// Mitsubishi GX Works2 project: EXAM2   PLC: Q03UDV

PROGRAM MAIN
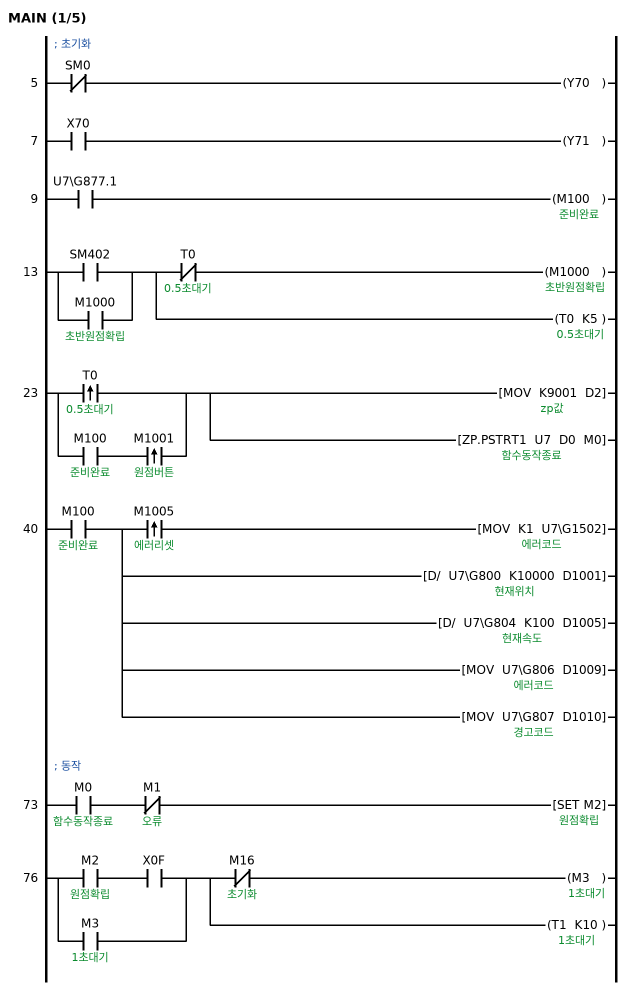
; 초기화
5     LDI     SM0
      OUT     Y70
7     LD      X70
      OUT     Y71
9     LD      U7\G877.1
      OUT     M100  ; 준비완료
13    LD      SM402
      OR      M1000  ; 초반원점확립
      MPS
      ANI     T0  ; 0.5초대기
      OUT     M1000  ; 초반원점확립
      MPP
      OUT     T0 K5  ; 0.5초대기
23    LDP     T0  ; 0.5초대기
      LD      M100  ; 준비완료
      ANDP    M1001  ; 원점버튼
      ORB
      MOV     K9001 D2  ; zp값
      ZP.PSTRT1 U7 D0 M0  ; 함수동작종료
40    LD      M100  ; 준비완료
      MPS
      ANDP    M1005  ; 에러리셋
      MOV     K1 U7\G1502  ; 에러코드
      MPP
      D/      U7\G800 K10000 D1001  ; 현재위치
      D/      U7\G804 K100 D1005  ; 현재속도
      MOV     U7\G806 D1009  ; 에러코드
      MOV     U7\G807 D1010  ; 경고코드
; 동작
73    LD      M0  ; 함수동작종료
      ANI     M1  ; 오류
      SET     M2  ; 원점확립
76    LD      M2  ; 원점확립
      AND     X0F
      OR      M3  ; 1초대기
      MPS
      ANI     M16  ; 초기화
      OUT     M3  ; 1초대기
      MPP
      OUT     T1 K10  ; 1초대기
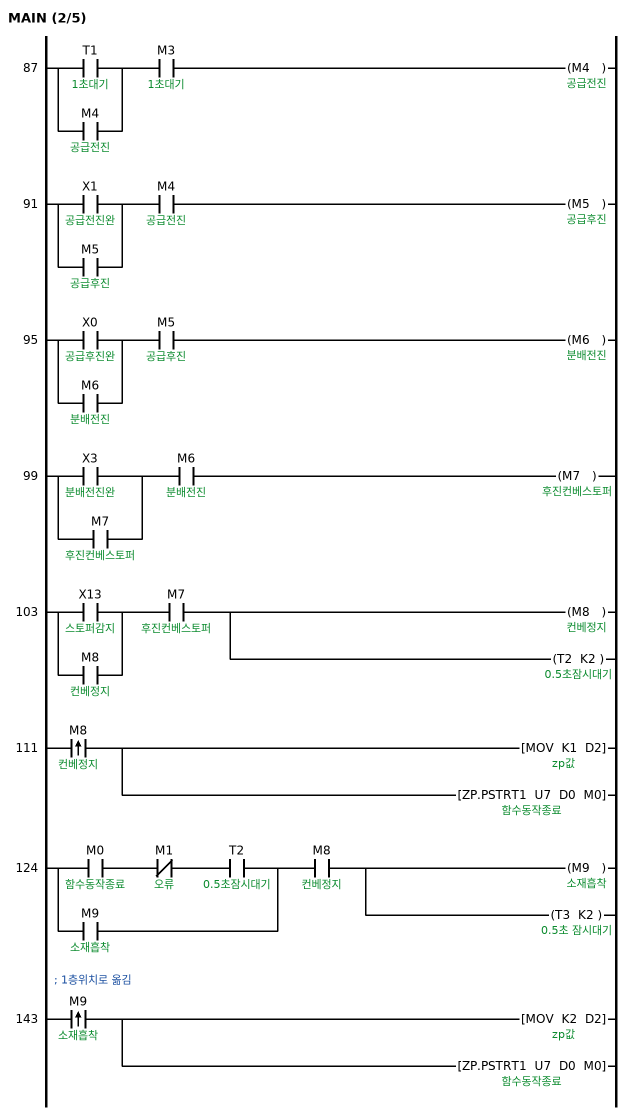
87    LD      T1  ; 1초대기
      OR      M4  ; 공급전진
      AND     M3  ; 1초대기
      OUT     M4  ; 공급전진
91    LD      X1  ; 공급전진완
      OR      M5  ; 공급후진
      AND     M4  ; 공급전진
      OUT     M5  ; 공급후진
95    LD      X0  ; 공급후진완
      OR      M6  ; 분배전진
      AND     M5  ; 공급후진
      OUT     M6  ; 분배전진
99    LD      X3  ; 분배전진완
      OR      M7  ; 후진컨베스토퍼
      AND     M6  ; 분배전진
      OUT     M7  ; 후진컨베스토퍼
103   LD      X13  ; 스토퍼감지
      OR      M8  ; 컨베정지
      AND     M7  ; 후진컨베스토퍼
      OUT     M8  ; 컨베정지
      OUT     T2 K2  ; 0.5초잠시대기
111   LDP     M8  ; 컨베정지
      MOV     K1 D2
      ZP.PSTRT1 U7 D0 M0
124   LD      M0  ; 함수동작종료
      ANI     M1  ; 오류
      AND     T2  ; 0.5초잠시대기
      OR      M9  ; 소재흡착
      AND     M8  ; 컨베정지
      OUT     M9  ; 소재흡착
      OUT     T3 K2  ; 0.5초 잠시대기
; 1층위치로 옮김
143   LDP     M9  ; 소재흡착
      MOV     K2 D2
      ZP.PSTRT1 U7 D0 M0
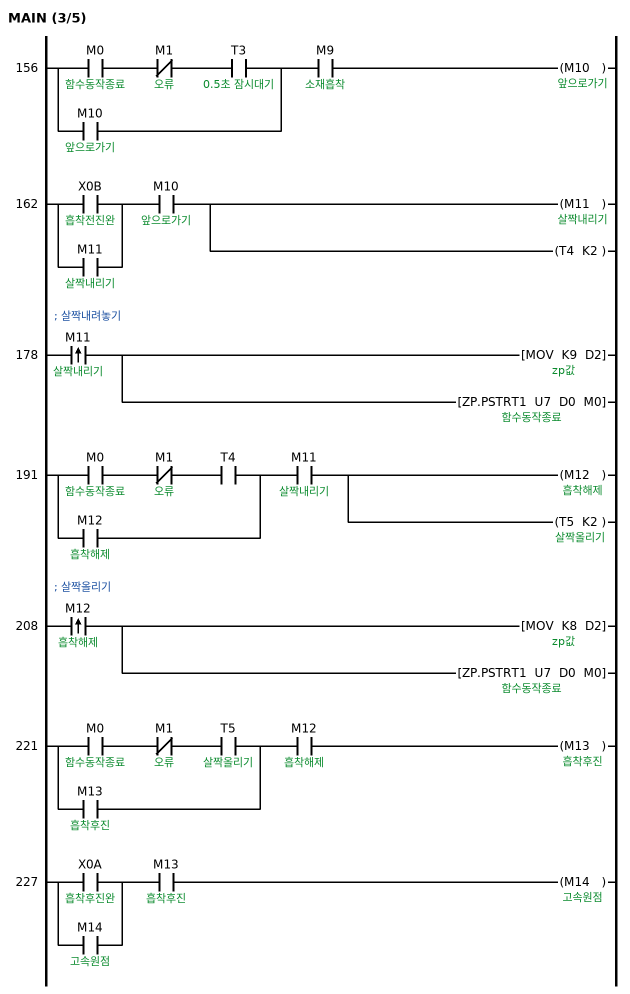
156   LD      M0  ; 함수동작종료
      ANI     M1  ; 오류
      AND     T3  ; 0.5초 잠시대기
      OR      M10  ; 앞으로가기
      AND     M9  ; 소재흡착
      OUT     M10  ; 앞으로가기
162   LD      X0B  ; 흡착전진완
      OR      M11  ; 살짝내리기
      AND     M10  ; 앞으로가기
      OUT     M11  ; 살짝내리기
      OUT     T4 K2
; 살짝내려놓기
178   LDP     M11  ; 살짝내리기
      MOV     K9 D2
      ZP.PSTRT1 U7 D0 M0
191   LD      M0  ; 함수동작종료
      ANI     M1  ; 오류
      AND     T4
      OR      M12  ; 흡착해제
      AND     M11  ; 살짝내리기
      OUT     M12  ; 흡착해제
      OUT     T5 K2  ; 살짝올리기
; 살짝올리기
208   LDP     M12  ; 흡착해제
      MOV     K8 D2
      ZP.PSTRT1 U7 D0 M0
221   LD      M0  ; 함수동작종료
      ANI     M1  ; 오류
      AND     T5  ; 살짝올리기
      OR      M13  ; 흡착후진
      AND     M12  ; 흡착해제
      OUT     M13  ; 흡착후진
227   LD      X0A  ; 흡착후진완
      OR      M14  ; 고속원점
      AND     M13  ; 흡착후진
      OUT     M14  ; 고속원점
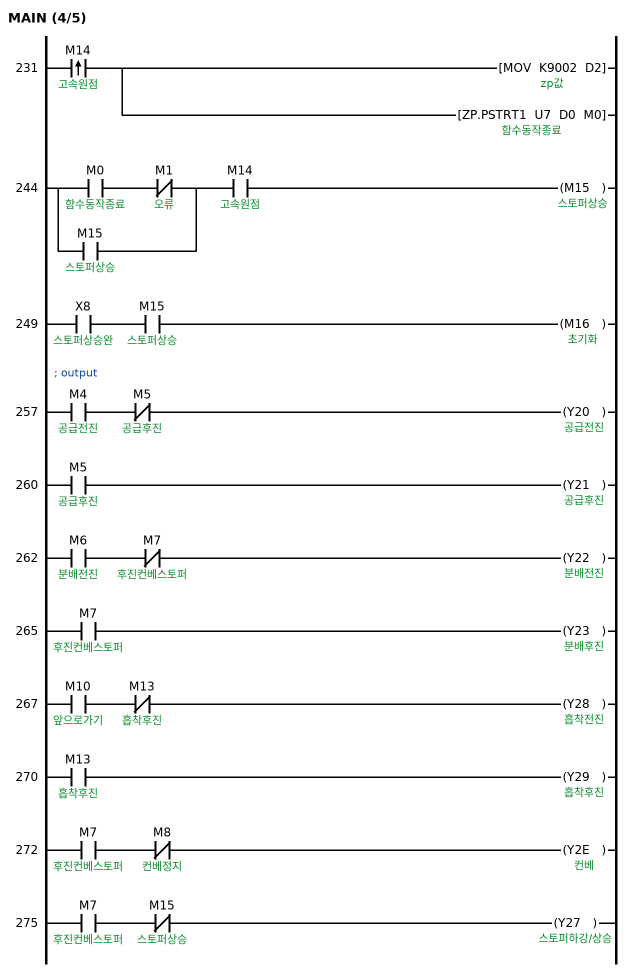
231   LDP     M14  ; 고속원점
      MOV     K9002 D2
      ZP.PSTRT1 U7 D0 M0
244   LD      M0  ; 함수동작종료
      ANI     M1  ; 오류
      OR      M15  ; 스토퍼상승
      AND     M14  ; 고속원점
      OUT     M15  ; 스토퍼상승
249   LD      X8  ; 스토퍼상승완
      AND     M15  ; 스토퍼상승
      OUT     M16  ; 초기화
; output
257   LD      M4  ; 공급전진
      ANI     M5  ; 공급후진
      OUT     Y20  ; 공급전진
260   LD      M5  ; 공급후진
      OUT     Y21  ; 공급후진
262   LD      M6  ; 분배전진
      ANI     M7  ; 후진컨베스토퍼
      OUT     Y22  ; 분배전진
265   LD      M7  ; 후진컨베스토퍼
      OUT     Y23  ; 분배후진
267   LD      M10  ; 앞으로가기
      ANI     M13  ; 흡착후진
      OUT     Y28  ; 흡착전진
270   LD      M13  ; 흡착후진
      OUT     Y29  ; 흡착후진
272   LD      M7  ; 후진컨베스토퍼
      ANI     M8  ; 컨베정지
      OUT     Y2E  ; 컨베
275   LD      M7  ; 후진컨베스토퍼
      ANI     M15  ; 스토퍼상승
      OUT     Y27  ; 스토퍼하강/상승
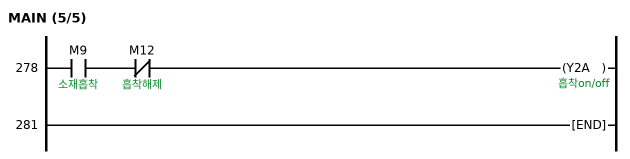
278   LD      M9  ; 소재흡착
      ANI     M12  ; 흡착해제
      OUT     Y2A  ; 흡착on/off
281   END
END_PROGRAM
